(* IEC 61131-3 sources: plc_generation_empirical_study/datasets/packages/internal_v0_1_precalibration_20260810/public_tasks/C06_M02_bounded_up_down_counter, 1 file *)

(* ---- interface.st ---- *)
FUNCTION_BLOCK C06_M02_bounded_up_down_counter
VAR_INPUT
    Add : BOOL;
    Remove : BOOL;
    Reset : BOOL;
    Capacity : INT;
END_VAR
VAR_OUTPUT
    Count : INT;
    Empty : BOOL;
    Full : BOOL;
    Conflict : BOOL;
END_VAR
END_FUNCTION_BLOCK
